// SIMATIC S7-200 project (STEP 7-Micro/WIN), CPU 224 REL 01.21

ORGANIZATION_BLOCK 主:OB1
TITLE=100t自动打包机新程序配触摸屏
// 
// 系统支持自动模式、手动模式和半自动模式三种操作模式，通过自动模式选择和手动模式选择在触摸屏上切换，模式显示实时反馈当前状态。
// 确保自动模式、手动模式和半自动模式互斥，同一时刻只能处于一种模式，避免操作冲突。
// 在自动模式下，按下自动起动按钮或通过自动起动中继触发自动起动，系统依次执行主缸前进压缩物料、穿线前进穿入打包线、结线正转缠绕线材、剪线下剪断线材等动作，最终完成打包。
// 主缸前进时，主缸前进保护约束要求主缸前限位为假，且穿线前进、穿线后退未动作，同时穿线后限位、剪线上限位、结线定位限位为真，主缸前进保护才允许动作，确保主缸不会因位置异常而受损。
// 穿线前进则受限于穿线前进保护约束，只有主缸前限位、剪线上限位、结线定位限位为真，且穿线前限位为假时，穿线前进保护才生效，保证穿线机构安全运行。
// 前进计数器记录主缸前进次数，达到前进计数预设值时触发主缸后退，避免超载。前进计数器应在打包完成后复位。
// 当自动起动且穿线后退动作时，触发打包完成。
// 手动模式下，操作员通过主缸前进按钮、穿线前进按钮、结线正转按钮等控制各部件动作。
// 按下主缸前进按钮可触发主缸前进，通过手动连续前进实现连续操作，但需满足主缸前进保护条件。
// 当急停按钮或急停触发时，所有输出（如主缸前进、穿线前进）和中间变量（如自动起动）立即复位，机器停止，确保操作员和设备安全。
// 定时器如主缸后退定时器、剪线延时1秒控制动作节奏，例如剪线下延时1秒后启动剪线上，保证剪线精准。
// 压力管理通过高压和低压切换，适应不同阶段需求。
// 打包总计数器和打包总数显示记录生产进度，自动时间设定定时器和自动时间显示确保周期一致。
// 
BEGIN
Network 1 // 网络题目 (单行)
//  
// 网络注释
//  
// 
LD     SM0.3
O      I0.0
O      M30.1
R      M0.0, 100
R      Q0.0, 30
R      M27.0, 40
Network 2 // 自动
// 
// 
LD     I0.2
AN     I0.3
O      M27.2
=      M0.0
Network 3 // 手动
// 
// 
LD     I0.3
AN     I0.2
O      M27.0
=      M0.1
Network 4 // 半自动
// 
// 
LDN    I0.2
AN     I0.3
A      M27.1
=      M0.2
Network 5 // 自动起动
// 
// 
LD     I0.1
O      M30.0
O      M0.4
O      M30.0
LD     M0.0
O      M0.2
ALD
AN     M30.1
AN     I0.0
=      M0.4
Network 6 // 后退等待起动
// 
// 
LD     T111
O      I2.1
O      M0.5
A      M0.0
AN     M0.2
A      M0.6
AN     M30.1
AN     I0.0
=      M0.5
Network 7 // 主缸前进保护m0.6
// 
// 
LDN    I3.0
AN     Q0.7
AN     Q1.0
A      I3.3
A      I3.5
A      I3.7
=      M0.6
Network 8 // 主缸后退保护m0.7
// 
// 
LDN    I3.1
AN     Q0.7
AN     Q1.0
A      I3.3
A      I3.5
A      I3.7
=      M0.7
Network 9 // 主缸前进Q0。3
// 
// 
LD     M0.4
EU
O      Q0.3
O      M0.5
A      M0.0
LD     M30.0
O      Q0.3
A      M0.2
OLD
A      M0.6
LD     M0.1
AN     M29.4
LD     I0.5
O      M28.0
ALD
O      M3.0
A      M0.6
OLD
=      Q0.3
Network 10 // 手动连续前进
// 
// 
LD     I0.5
O      M28.0
O      M3.0
A      M0.1
A      M29.4
AN     M30.1
AN     I0.0
AN     I3.0
=      M3.0
Network 11 // 主缸计数
// 
// 
LD     I3.0
LD     M0.0
O      M0.2
ALD
=      Q2.5
Network 12 // 主缸计数中继M1。0
// 
// 
LD     C10
O      M1.0
LD     M0.0
O      M0.2
ALD
AN     Q1.0
=      M1.0
Network 13 // 主缸后退Q0。4
// 
// 
LD     M0.4
LD     T101
O      T102
ALD
A      M0.7
AN     M1.0
LD     M0.1
LD     I0.6
O      M28.1
ALD
AN     M29.4
O      M3.1
A      M0.7
OLD
LPS
AN     I2.5
=      Q0.4
LPP
=      M5.0
Network 14 // 手动后退连续
// 
// 
LD     I0.6
O      M28.1
O      M3.1
AN     Q0.7
A      M0.1
A      M29.4
AN     M30.1
AN     I0.0
AN     I3.1
=      M3.1
Network 15 // 计数未到后退m1.1
// 
// 
LD     I3.0
O      M1.1
A      M0.7
AN     M1.0
=      M1.1
TON    T101, +15
Network 16 // 计数到达主缸后退加强保护定时器时间为穿线后退总时间
// 
// 
LD     Q1.0
TON    T107, +70
Network 17 // 计数到达后退t102
// 
// 
LD     I3.3
A      Q1.0
A      T107
EU
O      M1.2
AN     I3.1
A      M0.4
=      M1.2
TON    T102, +15
Network 18 // 泄压
// 
// 
LD     M1.1
O      M1.2
LD     M0.1
A      I0.7
A      M0.7
OLD
=      Q0.5
Network 19 // 自动时间设定
// 
// 
LD     Q0.4
ED
A      I3.1
LD     Q2.7
AN     I0.1
AN     M30.0
OLD
AN     M0.2
A      M0.0
AN     Q0.3
=      Q2.7
Network 20 // 穿线前进保护m1.3
// 
// 
LD     I3.0
A      I3.5
A      I3.7
AN     I3.2
=      M1.3
Network 21 // 穿线后退保护m1.4
// 
// 
LD     I3.0
A      I3.5
A      I3.7
AN     I3.3
=      M1.4
Network 22 // 穿线前进加强保护
// 
// 
LD     Q0.3
TON    T110, +10
Network 23 // 穿线前进Q0。7
// 
// 
LD     M1.0
O      Q0.7
LD     M0.0
O      M0.2
ALD
LDN    M29.4
A      M0.1
LD     M28.2
O      I1.2
ALD
OLD
O      M3.2
A      M1.3
=      Q0.7
Network 24 // 手动连续穿线
// 
// 
LD     I1.2
O      M28.2
O      M3.2
A      M0.1
A      M29.4
AN     M30.1
AN     I0.0
AN     I3.2
=      M3.2
Network 25 // 结线正转一圈所需时间
// 
// 
LD     Q0.7
ED
A      I3.2
LD     M0.0
O      M0.2
ALD
A      I3.0
EU
S      Q3.0, 1
Network 26
LD     Q3.0
O      M4.0
LPS
AN     T131
=      M4.0
LPP
TON    T131, +15
Network 27 // 结线正转一圈停止
// 
// 
LD     T131
EU
LD     I3.7
EU
OLD
RI     Q3.0, 1
Network 28 // 剪线起动
// 
// 
LD     Q3.0
LD     M0.0
O      M0.2
ALD
ED
S      M2.0, 1
Network 29 // 剪线延时1秒起动
// 
// 
LD     M2.0
TON    T103, +10
Network 30
LD     T103
EU
R      M2.0, 1
Network 31 // 开始剪线下
// 
// 
LD     T103
LD     M0.0
O      M0.2
ALD
LD     M0.1
LD     M29.0
O      I1.4
ALD
OLD
A      I3.0
A      I3.2
A      I3.7
EU
S      Q2.3, 1
Network 32 // 剪线下停止
// 
// 
LD     Q2.3
A      I3.4
EU
R      Q2.3, 1
Network 33 // 剪线上
// 
// 
LD     Q2.3
ED
S      M2.1, 1
Network 34 // 剪线延时1。5秒上
// 
// 
LD     M2.1
TON    T104, +15
Network 35 // 剪线上开始
// 
// 
LD     T104
=      Q2.4
Network 36 // 剪线上到位停止
// 
// 
LD     I3.5
R      M2.1, 1
Network 37 // 结线正转六圈起动
// 
// 
LD     Q2.4
LD     M0.0
O      M0.2
ALD
ED
S      M2.2, 1
Network 38 // 结线正转
// 
// 
LD     Q3.0
O      M2.2
LD     I1.5
O      M28.5
A      M0.1
OLD
A      I3.0
A      I3.2
AN     I2.4
=      Q0.1
Network 39 // 正转计数
// 
// 
LD     M0.2
O      M0.0
A      I3.7
A      Q0.1
LD     M0.0
O      M0.2
A      C1
EU
CTU    C1, +6
Network 40 // 正转六圈停
// 
// 
LD     C1
A      I3.7
R      M2.2, 1
Network 41 // 反转起动
// 
// 
LD     M2.2
ED
S      M2.3, 1
Network 42 // 反转延时一秒起动
// 
// 
LD     M2.3
TON    T105, +10
Network 43 // 反转开始
// 
// 
LD     M0.0
O      M0.2
A      T105
LD     M0.1
LD     I2.0
O      M28.4
ALD
OLD
A      I3.0
A      I3.2
AN     I2.4
=      Q0.2
Network 44 // 反转计数
// 
// 
LD     Q0.2
A      I3.7
LD     C2
EU
CTU    C2, +4
Network 45 // 反转停止
// 
// 
LD     C2
A      I3.7
R      M2.3, 1
R      Q0.2, 1
Network 46 // 穿线后退
// 
// 
LD     M0.0
O      M0.2
A      Q0.2
ED
S      M2.4, 1
Network 47 // 穿线延时一秒后退
// 
// 
LD     M2.4
TON    T106, +10
Network 48 // 穿线后退开始
// 
// 
LD     M0.0
O      M0.2
A      T106
LD     M0.1
AN     M29.4
LD     I1.3
O      M28.3
ALD
OLD
O      M3.3
A      I3.0
A      I3.5
A      I3.7
AN     I3.3
=      Q1.0
Network 49 // 手动穿线连续后退
// 
// 
LD     I1.3
O      M28.3
O      M3.3
A      M0.1
A      M29.4
AN     M30.1
AN     I0.0
AN     I3.3
=      M3.3
Network 50 // 穿线后退停止
// 
// 
LD     I3.3
R      M2.4, 1
Network 51 // 电磁溢流
// 
// 
LD     Q0.4
O      Q0.3
=      Q0.6
Network 52 // 泄压
// 
// 
LD     Q0.4
O      M5.0
=      Q0.5
Network 53 // 侧压夹紧
// 
// 
LD     I1.0
O      M28.6
=      Q1.1
Network 54 // 侧压放松
// 
// 
LD     I1.1
O      M28.7
=      Q2.0
Network 55 // 高压
// 
// 
LD     Q0.7
O      Q2.3
O      Q1.1
=      Q2.1
Network 56 // 低压
// 
// 
LD     Q1.0
O      Q2.4
O      Q2.0
=      Q2.2
Network 57 // 打包计数
// 
// 
LD     M0.4
A      Q1.0
EU
=      Q2.6
Network 58 // 主缸前限指示
// 
// 
LD     I3.0
=      Q3.1
Network 59 // 主缸后限指示
// 
// 
LD     I3.1
=      Q3.2
Network 60 // 穿线前限指示
// 
// 
LD     I3.2
=      Q3.3
Network 61 // 穿线后限指示
// 
// 
LD     I3.3
=      Q3.4
Network 62 // 结线定位指示
// 
// 
LD     I3.7
=      Q3.5
Network 63
// 辅助油泵起动
LD     Q0.7
O      Q1.0
O      Q1.1
O      Q2.0
O      Q2.3
O      Q2.4
=      Q0.0
Network 64
// 前进计数
LD     Q0.3
ED
A      I3.0
LD     T130
CTU    C10, VW20
Network 65
// 复位前进计数
LD     C10
TON    T130, +17
Network 66
// 前进计数显示
LD     M0.4
MOVW   C10, VW22
Network 67
// 自动时间设定
LD     Q2.7
TON    T111, VW100
Network 68
LD     SM0.0
MOVW   VW112, VW28
/I     +10, VW28
Network 69
// 自动时间显示
LD     Q2.7
MOVW   T111, VW112
Network 70
// 打包总计数
LD     Q2.6
LD     M29.2
CTU    C11, +9999
Network 71
LD     SM0.0
MOVW   VW30, VW100
*I     +10, VW100
Network 72
// 打包总数显示
LD     SM0.0
MOVW   C11, VW26
Network 73
// 手动
LD     SM0.0
AW=    VW24, +0
=      M27.0
Network 74
// 半自动
LD     SM0.0
AW=    VW24, +1
=      M27.1
Network 75
// 自动
LD     SM0.0
AW=    VW24, +2
=      M27.2
END_ORGANIZATION_BLOCK
